FUNCTION fnLogMsgInit : BOOL
VAR_INPUT
		//logMsgPtr : REFERENCE TO LogMsg;
		logMsgPtr 		 : POINTER TO LogMsg;
		category  		 : STRING[LOG_MSG_CATEGORY_LENGTH];
		globalArrayAddr  : POINTER TO LogGlobalArrayObj;
		encoderAngleAddr : POINTER TO REAL;	
END_VAR
VAR
	
END_VAR

	fnLogMsgInit := logMsgPtr^.InitLogger(category, globalArrayAddr, encoderAngleAddr);

END_FUNCTION

(* stored: Version 1.1.0.1, ProductVersion 3.1.4024.3
   POU fnLogMsgInit: Id {808e14e6-a536-0bd1-0008-2051819acd95}, SpecialFunc None *)
